// TIA Portal project "LearningFactory_4_0_24V_Task05_VacuumGripperVGR_V18" (V18)

(* hardware
DEVICE "ET 200SP-Station_1"  ET 200SP-Station
   slot 0: "Baugruppenträger_0"  Rack  6ES5 710-8MAx1
   slot 1: "PLC"  CPU 1512SP F-1 PN  6ES7 512-1SK01-0AB0  V2.8
      slot 32768: "PROFINET"  X1
   slot 2: "DO1+2"  DQ 16x24VDC/0.5A ST  6ES7 132-6BH01-0BA0  V0.0
      slot 1: "DO1+2"  DQ 16x24VDC/0.5A ST
   slot 3: "DO3+4"  DQ 16x24VDC/0.5A ST  6ES7 132-6BH01-0BA0  V0.0
      slot 1: "DO3+4"  DQ 16x24VDC/0.5A ST
   slot 4: "DO5+6"  DQ 16x24VDC/0.5A ST  6ES7 132-6BH01-0BA0  V0.0
      slot 1: "DO5+6"  DQ 16x24VDC/0.5A ST
   slot 5: "DO7-14"  DQ 4x24VDC/2A HS  6ES7 132-6BD20-0DA0  V2.0
      slot 1: "DO7-14"  DQ 4x24VDC/2A HS
   slot 6: "DO15-22"  DQ 4x24VDC/2A HS  6ES7 132-6BD20-0DA0  V2.0
      slot 1: "DO15-22"  DQ 4x24VDC/2A HS
   slot 7: "DO23-30"  DQ 4x24VDC/2A HS  6ES7 132-6BD20-0DA0  V2.0
      slot 1: "DO23-30"  DQ 4x24VDC/2A HS
   slot 8: "DI1+2"  DI 16x24VDC ST  6ES7 131-6BH01-0BA0  V0.0
      slot 1: "DI1+2"  DI 16x24VDC ST
   slot 9: "DI3+4"  DI 16x24VDC ST  6ES7 131-6BH01-0BA0  V0.0
      slot 1: "DI3+4"  DI 16x24VDC ST
   slot 10: "DI5"  DI 8x24VDC HS  6ES7 131-6BF00-0DA0  V1.0
      slot 1: "DI5"  DI 8x24VDC HS
   slot 11: "DI6"  DI 8x24VDC HS  6ES7 131-6BF00-0DA0  V1.0
      slot 1: "DI6"  DI 8x24VDC HS
   slot 12: "AI7-10"  AI 2xU ST  6ES7 134-6FB00-0BA1  V1.0
      slot 1: "AI7-10"  AI 2xU ST
   slot 13: "End"  Server module  6ES7 193-6PA00-0AA0  V1.1
      slot 1: "End"  Server module
   slot 127: "BA 2xRJ45"  BA 2xRJ45  6ES7 193-6AR00-0AA0  V0.0
      slot 32769: "Port_1"  6ES7 193-6AR00-0AA0
      slot 32770: "Port_2"  6ES7 193-6AR00-0AA0
*)

// ===== PLC "PLC"  CPU 1512SP F-1 PN =====

VAR_GLOBAL   // PLC tag table "Start_Stop"
   "IX_START" AT %I4.4 : Bool;
   "IX_STOP" AT %I4.6 : Bool;
END_VAR

VAR_GLOBAL   // PLC tag table "VGR - Vacuum Gripper Robot"
   "IX_VGR_RefSwitchVerticalAxis_I1" AT %I1.6 : Bool;
   "IX_VGR_RefSwitchHorizontalAxis_I2" AT %I3.6 : Bool;
   "IX_VGR_RefSwitchRotate_I3" AT %I3.7 : Bool;
   "IX_VGR_EncoderVerticalAxisImp1_B1" AT %I6.0 : Bool;
   "IX_VGR_EncoderVerticalAxisImp2_B2" AT %I6.4 : Bool;
   "IX_VGR_EncoderHorizontalAxisImp1_B3" AT %I6.1 : Bool;
   "IX_VGR_EncoderHorizontalAxisImp2_B4" AT %I6.5 : Bool;
   "IX_VGR_EncoderRotateImp1_B5" AT %I6.2 : Bool;
   "IX_VGR_EncoderRotateImp2_B6" AT %I6.6 : Bool;
   "QX_VGR_M1_VerticalAxisUp_Q1" AT %Q2.0 : Bool;
   "QX_VGR_M1_VerticalAxisDown_Q2" AT %Q2.1 : Bool;
   "QX_VGR_M2_HorizontalAxisBackward_Q3" AT %Q2.2 : Bool;
   "QX_VGR_M2_HorizontalAxisForward_Q4" AT %Q2.3 : Bool;
   "QX_VGR_M3_RotateClockwise_Q5" AT %Q2.4 : Bool;
   "QX_VGR_M3_RotateCounterclockwise_Q6" AT %Q2.5 : Bool;
   "QX_VGR_Compressor_Q7" AT %Q2.6 : Bool;
   "QX_VGR_ValveVacuum_Q8" AT %Q2.7 : Bool;
   "QW_VGR_PWM_Vertical_M1" AT %QW15 : Int;
   "QW_VGR_PWM_Horizontal_M2" AT %QW17 : Int;
   "QW_VGR_PWM_Rotate_M3" AT %QW19 : Int;
END_VAR

DATA_BLOCK "Task05_VacuumGripper_DB"   // DB3
{ S7_Optimized_Access := 'TRUE' }
VERSION : 0.1
// stored: InstanceOfName Task05_VacuumGripper
"Task05_VacuumGripper"
BEGIN
END_DATA_BLOCK

FUNCTION_BLOCK "Task05_VacuumGripper"   // FB3, SCL
{ S7_Optimized_Access := 'TRUE' }
VERSION : 0.1
   VAR_INPUT
      Start : Bool;
      Stop : Bool;
      RefSwitchRotate : Bool;
      RefSwitchVerticalAxis : Bool;
      RefSwitchHorizontalAxis : Bool;
      EncoderVerticalAxisImp1 : Bool;
      EncoderRotateImp1 : Bool;
   END_VAR
   VAR_OUTPUT
      M1_VerticalAxisDown : Bool;
      M1_VerticalAxisUp : Bool;
      PWM_Vertical : Int;
      M2_HorizontalAxisBackward : Bool;
      M2_HorizontalAxisForward : Bool;
      PWM_Horizontal : Int;
      M3_RotateClockwise : Bool;
      M3_RotateCounterclockwise : Bool;
      PWM_Rotate : Int;
      ValveVacuum : Bool;
      Compressor : Bool;
   END_VAR
   VAR
      Step_number : Int;
      PositioningCounterVertical : Int;
      PositioningCounterRotate : Int;
      R_TRIG_PulseCountVertical : R_TRIG;
      R_TRIG_PulseCountRotate : R_TRIG;
      IEC_Timer_VacuumOn : TON_TIME;
      IEC_Timer_VacuumOff : TON_TIME;
   END_VAR
BEGIN

   // Reset sequencer with pushbutton STOP 
   // Rücksetzen der Schrittkette  mit Taster STOP

   IF #Stop THEN
       #Step_number := 0;
   END_IF;

   // Start sequencer with pushbutton START
   // Starten der Schrittkette  mit Taster START

   CASE #Step_number OF
       0:  // Initial step 1 / Initialschritt 1
           #M1_VerticalAxisDown := FALSE;          //Vertical axis down off / Vertikale Achse runterfahren aus
           #M1_VerticalAxisUp := FALSE;            //Vertical axis up off/ Vertikale Achse hochfahren aus
           #M2_HorizontalAxisBackward := FALSE;    //Horizontal axis back off/ Horizontale Achse zurückfahren aus    
           #M2_HorizontalAxisForward := FALSE;     //Horizontal axis back off/ Horizontale Achse zurückfahren aus  
           #M3_RotateClockwise := FALSE;           // Rotation clockwise off / Rotation im Uhrzeigersinnaus aus
           #M3_RotateCounterclockwise := FALSE;    // Rotation counter clockwise off/ Rotation gegen den Uhrzeigersinn aus
           #ValveVacuum := FALSE;                  // Vacuum gripper off / Vakuumgreifer aus
           #Compressor := FALSE;                   // Compressor oiff / Kompressor oiff
           #PWM_Vertical := 400;                   // PWM-signal vertical axis / PWM-Signal vertikale Achse
           #PWM_Horizontal := 400;                 //PWM-signal horizontal axis / PWM-Signal vertikae Achse
           #PWM_Rotate := 400;                     //PWM-signal rotation / PWM-Signal Rotation
           #PositioningCounterVertical := 0;       //reset positioning counter vertical axis / Positionszähler zurücksetzen vertikale Achse
           #PositioningCounterRotate := 0;         //reset positioning counter rotation / Positionszähler zurücksetzen Rotation
           RESET_TIMER(#IEC_Timer_VacuumOn);       // Reset timer to pick workpiece / Rücksetzen des Timers um das Werkstück aufzunehmen
           RESET_TIMER(#IEC_Timer_VacuumOff);      // Reset timer to drop workpiece / Rücksetzen des Timers um das Werkstück abzulegen

           IF #Start THEN
               #Step_number := #Step_number + 1;
           END_IF;

       1:  // Step 1 move back horizontal axis / Schritt 1 horizontale Ache einfahren
           #M2_HorizontalAxisBackward := TRUE;     //Horizontal axis back / Horizontale Achse zurückfahren   

           IF #RefSwitchHorizontalAxis THEN
               #Step_number := #Step_number + 1;
           END_IF;

       2:  // Step 2 move up vertical axis / Schritt 2 vertikale Achse nach oben fahren
           #M2_HorizontalAxisBackward := FALSE; //Horizontal axis back off / Horizontale Achse zurückfahren aus   
           #M1_VerticalAxisUp := TRUE;          //Vertical axis up / Vertikale Achse hochfahren 

           IF  #RefSwitchVerticalAxis  THEN
               #Step_number := #Step_number + 1;
           END_IF;

       3:  // Step 3 rotation clockwisec/ Schritt 3 Rotation im Uhrzeigersinn
           #M1_VerticalAxisUp := FALSE;        //Vertical axis up off / Vertikale Achse hochfahren aus
           #M3_RotateClockwise := TRUE;        //Rotation clockwise / Rotation im Uhrzeigersinn
           #PositioningCounterVertical := 0;   //reset positioning counter vertical axis / Positionszähler zurücksetzen vertikale Achse

           IF  #RefSwitchRotate  THEN
               #Step_number := #Step_number + 1;
           END_IF;

       4:  // Step 4 move down vertical axis; start positioning counter / Schritt 4  abwärts vertikale Achse; Zähler zum Positionieren starten
           #M3_RotateClockwise := False;       //Rotation clockwise off / Rotation im Uhrzeigersinn aus
           #M1_VerticalAxisDown := TRUE;       //Vertical axis down / Vertikale Achse runterfahren 
           #R_TRIG_PulseCountVertical(CLK:=#EncoderVerticalAxisImp1); // Positive edge detection encoder vertical / Positive Flanke an Encoder vertikal
           IF #R_TRIG_PulseCountVertical.Q THEN
               #PositioningCounterVertical := #PositioningCounterVertical + 1;  // Positioning Counter +1 / Zähler zum Positionieren +1
           END_IF;

           IF #PositioningCounterVertical >= 170 THEN
               #Step_number := #Step_number + 1;
           END_IF;

       5:  // Step 5 vacuum on / Schritt 5 Vakuum einschalten
           #M1_VerticalAxisDown := FALSE;      //Vertical axis down off / Vertikale Achse runterfahren aus
           #PositioningCounterVertical := 0;   //reset positioning counter vertical axis / Positionszähler zurücksetzen vertikale Achse
           #ValveVacuum := TRUE;               // Vacuum gripper on / Vakuumgreifer ein
           #Compressor := TRUE;                // Compressor on / Kompressor ein
           #IEC_Timer_VacuumOn(IN:=#ValveVacuum, // Start Timer to pick workpiece / Timer starten um das Werkstück aufzunehmen
                       PT:=T#2s);

           IF #IEC_Timer_VacuumOn.Q THEN
               #Step_number := #Step_number + 1;
           END_IF;

       6:  // Step 6 move up vertical axis / Schritt 6 vertikale Achse nach oben fahren
           #M1_VerticalAxisUp := TRUE;         //Vertical axis up / Vertikale Achse hochfahren 
           #PositioningCounterRotate := 0;     //reset positioning counter rotation / Positionszähler zurücksetzen Rotation
           RESET_TIMER(#IEC_Timer_VacuumOn);   // Reset timer to pick workpiece / Rücksetzen des Timers um das Werkstück aufzunehmen

           IF #RefSwitchVerticalAxis THEN
               #Step_number := #Step_number + 1;
           END_IF;

       7:  // Step 7 Rotation counter clockwise; start positioning counter / Schritt 7 Rotation gegen den Uhrzeigersinn; Zähler zum Positionieren starten
           #M1_VerticalAxisUp := FALSE;                //Vertical axis up off / Vertikale Achse hochfahren aus 
           #M3_RotateCounterclockwise := TRUE;         //Rotation counter clockwise / Rotation gegen Uhrzeigersinn
           #PositioningCounterVertical := 0;           //reset positioning counter vertical axis / Positionszähler zurücksetzen vertikale Achse
           #R_TRIG_PulseCountRotate(CLK := #EncoderRotateImp1); // Positive edge detection encoder rotation / Positive Flanke an Encoder Rotation
           IF #R_TRIG_PulseCountRotate.Q THEN
               #PositioningCounterRotate := #PositioningCounterRotate + 1;  // Positioning Counter +1 / Zähler zum Positionieren +1
           END_IF;
           IF #PositioningCounterRotate >= 116 THEN
               #Step_number := #Step_number + 1;
           END_IF;

       8:  // Step 8 move down vertical axis; start positioning counter / Schritt 8  abwärts vertikale Achse; Zähler zum Positionieren starten
           #M3_RotateCounterclockwise := False;       //Rotation counter clockwise off / Rotation gegen Uhrzeigersinn aus
           #PositioningCounterRotate := 0;             //reset positioning counter rotation / Positionszähler zurücksetzen Rotation
           #M1_VerticalAxisDown := TRUE;               //Vertical axis down / Vertikale Achse runterfahren 
           #R_TRIG_PulseCountVertical(CLK := #EncoderVerticalAxisImp1); // Positive edge detection encoder vertical / Positive Flanke an Encoder vertikal
           IF #R_TRIG_PulseCountVertical.Q THEN
               #PositioningCounterVertical := #PositioningCounterVertical + 1;  // Positioning Counter +1 / Zähler zum Positionieren +1
           END_IF;

           IF #PositioningCounterVertical >= 165 THEN
               #Step_number := #Step_number + 1;
           END_IF;

       9:  // Step 5 vacuum off / Schritt 9 Vakuum ausschalten
           #M1_VerticalAxisDown := FALSE;      //Vertical axis down off / Vertikale Achse runterfahren aus
           #PositioningCounterVertical := 0;   //reset positioning counter vertical axis / Positionszähler zurücksetzen vertikale Achse
           #ValveVacuum := FALSE;               // Vacuum gripper off / Vakuumgreifer aus
           #Compressor := FALSE;                // Compressor off / Kompressor aus
           #IEC_Timer_VacuumOff(IN := NOT #ValveVacuum,  // Start Timer to drop workpiece / Timer starten um das Werkstück abzulegen
                               PT := T#2s);

          IF #IEC_Timer_VacuumOff.Q THEN
              #Step_number := 0;
          END_IF;

       ELSE  // Statement section ELSE
           ;
   END_CASE;
END_FUNCTION_BLOCK

ORGANIZATION_BLOCK "Main"   // OB1, SCL, ProgramCycle
TITLE = "Main Program Sweep (Cycle)"
{ S7_Optimized_Access := 'TRUE' }
VERSION : 0.1
   VAR_INPUT
      Initial_Call : Bool;   // Initial call of this OB
      Remanence : Bool;   // =True, if remanent data are available
   END_VAR
BEGIN


   // Call subroutine VacuumGripper
   // Aufruf Unterprogramm VacuumGripper

   "Task05_VacuumGripper_DB"(Start:="IX_START",
                             Stop:= NOT "IX_STOP",
                             RefSwitchRotate:="IX_VGR_RefSwitchRotate_I3",
                             RefSwitchVerticalAxis:="IX_VGR_RefSwitchVerticalAxis_I1",
                             RefSwitchHorizontalAxis:="IX_VGR_RefSwitchHorizontalAxis_I2",
                             EncoderVerticalAxisImp1:="IX_VGR_EncoderVerticalAxisImp1_B1",
                             EncoderRotateImp1:="IX_VGR_EncoderRotateImp1_B5",
                             M1_VerticalAxisDown=>"QX_VGR_M1_VerticalAxisDown_Q2",
                             M1_VerticalAxisUp=>"QX_VGR_M1_VerticalAxisUp_Q1",
                             PWM_Vertical=>"QW_VGR_PWM_Vertical_M1",
                             M2_HorizontalAxisBackward=>"QX_VGR_M2_HorizontalAxisBackward_Q3",
                             M2_HorizontalAxisForward=>"QX_VGR_M2_HorizontalAxisForward_Q4",
                             PWM_Horizontal=>"QW_VGR_PWM_Horizontal_M2",
                             M3_RotateClockwise=>"QX_VGR_M3_RotateClockwise_Q5",
                             M3_RotateCounterclockwise=>"QX_VGR_M3_RotateCounterclockwise_Q6",
                             PWM_Rotate=>"QW_VGR_PWM_Rotate_M3",
                             ValveVacuum=>"QX_VGR_ValveVacuum_Q8",
                             Compressor=>"QX_VGR_Compressor_Q7");
END_ORGANIZATION_BLOCK